// TIA Portal V19 export
FUNCTION "TEST_O_TODO_Fun" : Void   // FC200, LAD
// stored: SetENOAutomatically false
   VAR_TEMP   // added for the SCL form of the ladder/FBD networks
      _w1 : Bool;
   END_VAR
BEGIN

REGION Network 1
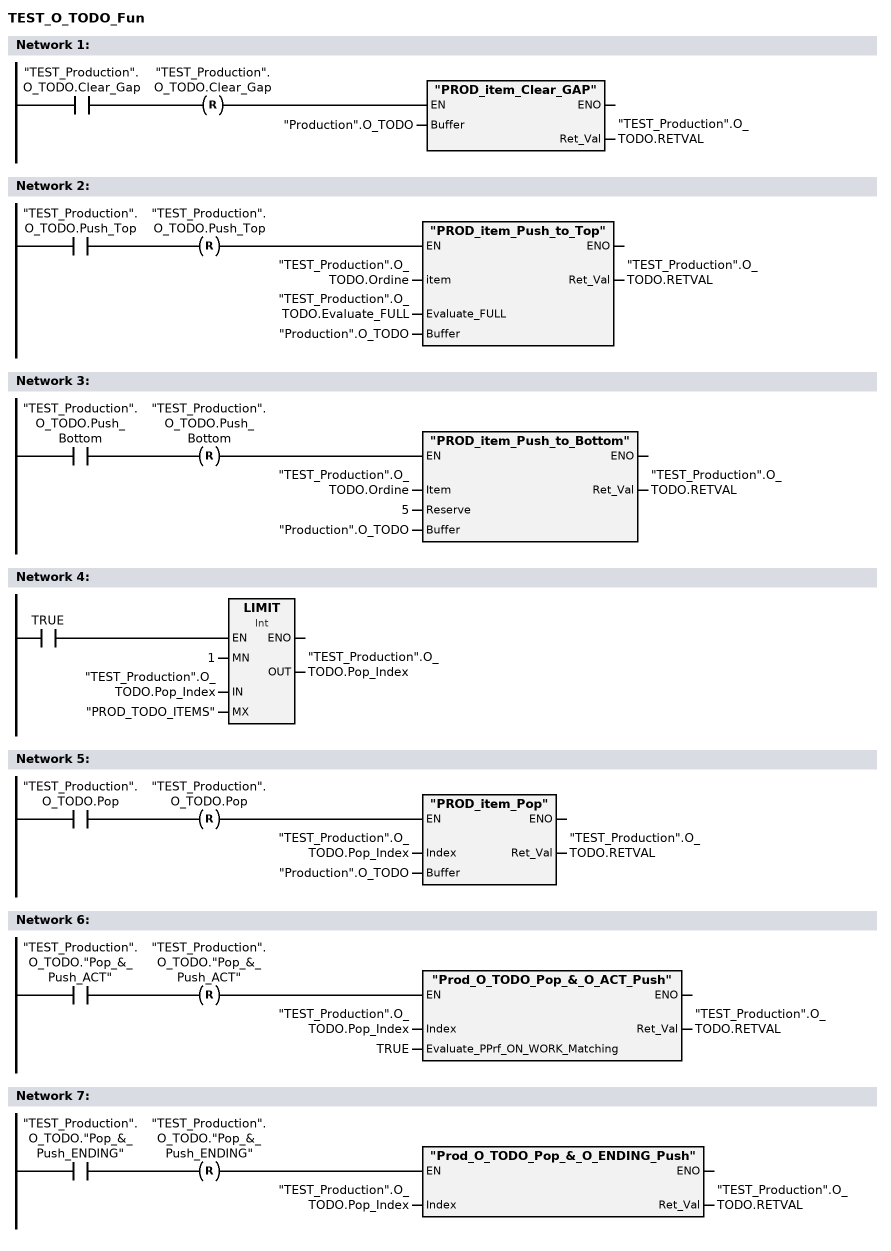
   RUNG wire#powerrail
      Contact( "TEST_Production".O_TODO.Clear_Gap )
      R_Coil( "TEST_Production".O_TODO.Clear_Gap )
      "PROD_item_Clear_GAP"(Buffer := "Production".O_TODO, Ret_Val => "TEST_Production".O_TODO.RETVAL)
   END_RUNG
   // the same network as SCL:
   #_w1 := "TEST_Production".O_TODO.Clear_Gap;
   IF #_w1 THEN
       "TEST_Production".O_TODO.Clear_Gap := FALSE;
       "TEST_Production".O_TODO.RETVAL := "PROD_item_Clear_GAP"(Buffer := "Production".O_TODO);
   END_IF;
END_REGION

REGION Network 2
   RUNG wire#powerrail
      Contact( "TEST_Production".O_TODO.Push_Top )
      R_Coil( "TEST_Production".O_TODO.Push_Top )
      "PROD_item_Push_to_Top"(item := "TEST_Production".O_TODO.Ordine, Evaluate_FULL := "TEST_Production".O_TODO.Evaluate_FULL, Buffer := "Production".O_TODO, Ret_Val => "TEST_Production".O_TODO.RETVAL)
   END_RUNG
   // the same network as SCL:
   #_w1 := "TEST_Production".O_TODO.Push_Top;
   IF #_w1 THEN
       "TEST_Production".O_TODO.Push_Top := FALSE;
       "TEST_Production".O_TODO.RETVAL := "PROD_item_Push_to_Top"(item := "TEST_Production".O_TODO.Ordine,
                               Evaluate_FULL := "TEST_Production".O_TODO.Evaluate_FULL,
                               Buffer := "Production".O_TODO);
   END_IF;
END_REGION

REGION Network 3
   RUNG wire#powerrail
      Contact( "TEST_Production".O_TODO.Push_Bottom )
      R_Coil( "TEST_Production".O_TODO.Push_Bottom )
      "PROD_item_Push_to_Bottom"(Item := "TEST_Production".O_TODO.Ordine, Reserve := 5, Buffer := "Production".O_TODO, Ret_Val => "TEST_Production".O_TODO.RETVAL)
   END_RUNG
   // the same network as SCL:
   #_w1 := "TEST_Production".O_TODO.Push_Bottom;
   IF #_w1 THEN
       "TEST_Production".O_TODO.Push_Bottom := FALSE;
       "TEST_Production".O_TODO.RETVAL := "PROD_item_Push_to_Bottom"(Item := "TEST_Production".O_TODO.Ordine,
                               Reserve := 5,
                               Buffer := "Production".O_TODO);
   END_IF;
END_REGION

REGION Network 4
   RUNG wire#powerrail
      Contact( TRUE )
      { S7_Templates := "value_type := Int" } Limit(mn := 1, in := "TEST_Production".O_TODO.Pop_Index, mx := "PROD_TODO_ITEMS", out => "TEST_Production".O_TODO.Pop_Index)
   END_RUNG
   // the same network as SCL:
   IF TRUE THEN
       "TEST_Production".O_TODO.Pop_Index := LIMIT(MN := 1, IN := "TEST_Production".O_TODO.Pop_Index, MX := "PROD_TODO_ITEMS");
   END_IF;
END_REGION

REGION Network 5
   RUNG wire#powerrail
      Contact( "TEST_Production".O_TODO.Pop )
      R_Coil( "TEST_Production".O_TODO.Pop )
      "PROD_item_Pop"(Index := "TEST_Production".O_TODO.Pop_Index, Buffer := "Production".O_TODO, Ret_Val => "TEST_Production".O_TODO.RETVAL)
   END_RUNG
   // the same network as SCL:
   #_w1 := "TEST_Production".O_TODO.Pop;
   IF #_w1 THEN
       "TEST_Production".O_TODO.Pop := FALSE;
       "TEST_Production".O_TODO.RETVAL := "PROD_item_Pop"(Index := "TEST_Production".O_TODO.Pop_Index,
                               Buffer := "Production".O_TODO);
   END_IF;
END_REGION

REGION Network 6
   RUNG wire#powerrail
      Contact( "TEST_Production".O_TODO."Pop_&_Push_ACT" )
      R_Coil( "TEST_Production".O_TODO."Pop_&_Push_ACT" )
      "Prod_O_TODO_Pop_&_O_ACT_Push"(Index := "TEST_Production".O_TODO.Pop_Index, Evaluate_PPrf_ON_WORK_Matching := TRUE, Ret_Val => "TEST_Production".O_TODO.RETVAL)
   END_RUNG
   // the same network as SCL:
   #_w1 := "TEST_Production".O_TODO."Pop_&_Push_ACT";
   IF #_w1 THEN
       "TEST_Production".O_TODO."Pop_&_Push_ACT" := FALSE;
       "TEST_Production".O_TODO.RETVAL := "Prod_O_TODO_Pop_&_O_ACT_Push"(Index := "TEST_Production".O_TODO.Pop_Index,
                               Evaluate_PPrf_ON_WORK_Matching := TRUE);
   END_IF;
END_REGION

REGION Network 7
   RUNG wire#powerrail
      Contact( "TEST_Production".O_TODO."Pop_&_Push_ENDING" )
      R_Coil( "TEST_Production".O_TODO."Pop_&_Push_ENDING" )
      "Prod_O_TODO_Pop_&_O_ENDING_Push"(Index := "TEST_Production".O_TODO.Pop_Index, Ret_Val => "TEST_Production".O_TODO.RETVAL)
   END_RUNG
   // the same network as SCL:
   #_w1 := "TEST_Production".O_TODO."Pop_&_Push_ENDING";
   IF #_w1 THEN
       "TEST_Production".O_TODO."Pop_&_Push_ENDING" := FALSE;
       "TEST_Production".O_TODO.RETVAL := "Prod_O_TODO_Pop_&_O_ENDING_Push"(Index := "TEST_Production".O_TODO.Pop_Index);
   END_IF;
END_REGION
END_FUNCTION
